// TIA Portal project "Carroponte" (V15.1)

(* hardware
DEVICE "S7-1200 station_1"  S7-1200 Station
   slot 0: "Telaio di montaggio_0"  S7-1200 Rack  Rack  V1.0
   slot 1: "PLC_1"  CPU 1214C DC/DC/DC  6ES7 214-1AG40-0XB0  V4.2
*)

// ===== PLC "PLC_1"  CPU 1214C DC/DC/DC =====

VAR_GLOBAL   // PLC tag table "Tabella delle variabili standard"
   "right" AT %Q0.0 : Bool;
   "left" AT %Q0.1 : Bool;
   "up" AT %Q0.2 : Bool;
   "down" AT %Q0.3 : Bool;
   "start" AT %I0.0 : Bool;
   "s1" AT %I0.1 : Bool;
   "s2" AT %I0.2 : Bool;
   "s3" AT %I0.3 : Bool;
   "sup" AT %I0.4 : Bool;
   "sdown" AT %I0.5 : Bool;
END_VAR

VAR_GLOBAL CONSTANT   // PLC tag table "Tabella delle variabili standard"
   "tempo" : Time := T#5s;
END_VAR

DATA_BLOCK "Variabili_Stato"   // DB1
{ S7_Optimized_Access := 'TRUE' }
VERSION : 0.1
   VAR RETAIN
      home : Bool := true;
   END_VAR
   VAR
      destra1 : Bool;
      su : Bool;
      destra2 : Bool;
      attesa : Bool;
      sinistra : Bool;
      giu : Bool;
   END_VAR
BEGIN
END_DATA_BLOCK

// folder: System blocks/Program resources

DATA_BLOCK "IEC_Timer_0_DB"   // DB2
{ S7_Optimized_Access := 'TRUE' }
AUTHOR : Simatic
FAMILY : IEC
NAME : IEC_TMR
VERSION : 1.0
// stored: InstanceOfName IEC_TIMER
"IEC_TIMER"
BEGIN
END_DATA_BLOCK

// folder: (top level)

ORGANIZATION_BLOCK "Main"   // OB1, LAD, ProgramCycle
TITLE = "Main Program Sweep (Cycle)"
{ S7_Optimized_Access := 'TRUE' }
VERSION : 0.1
   VAR_INPUT
      Initial_Call : Bool;   // Initial call of this OB
      Remanence : Bool;   // =True, if remanent data are available
   END_VAR
BEGIN

REGION Network 1
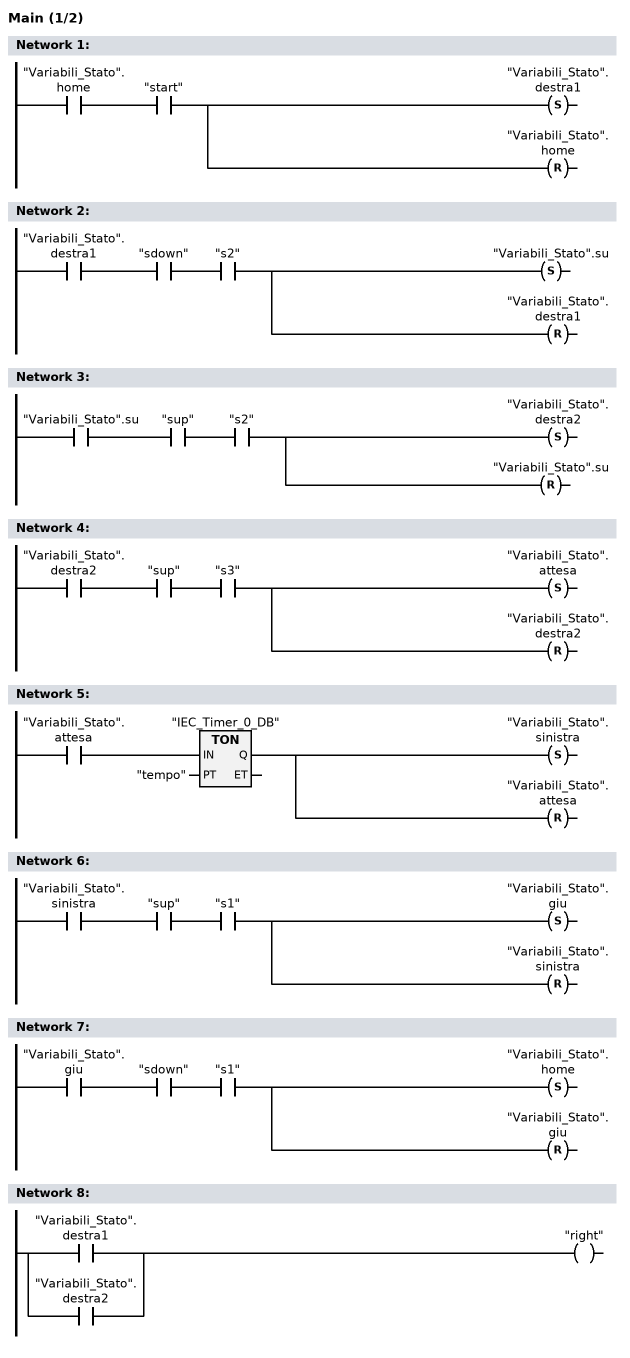
   RUNG wire#powerrail
      Contact( "Variabili_Stato".home )
      Contact( "start" )
      wire#w1
      S_Coil( "Variabili_Stato".destra1 )
   END_RUNG
   RUNG wire#w1
      R_Coil( "Variabili_Stato".home )
   END_RUNG
   // the same network as SCL:
   IF "Variabili_Stato".home AND "start" THEN
       "Variabili_Stato".destra1 := TRUE;
       "Variabili_Stato".home := FALSE;
   END_IF;
END_REGION

REGION Network 2
   RUNG wire#powerrail
      Contact( "Variabili_Stato".destra1 )
      Contact( "sdown" )
      Contact( "s2" )
      wire#w1
      S_Coil( "Variabili_Stato".su )
   END_RUNG
   RUNG wire#w1
      R_Coil( "Variabili_Stato".destra1 )
   END_RUNG
   // the same network as SCL:
   IF "Variabili_Stato".destra1 AND "sdown" AND "s2" THEN
       "Variabili_Stato".su := TRUE;
       "Variabili_Stato".destra1 := FALSE;
   END_IF;
END_REGION

REGION Network 3
   RUNG wire#powerrail
      Contact( "Variabili_Stato".su )
      Contact( "sup" )
      Contact( "s2" )
      wire#w1
      S_Coil( "Variabili_Stato".destra2 )
   END_RUNG
   RUNG wire#w1
      R_Coil( "Variabili_Stato".su )
   END_RUNG
   // the same network as SCL:
   IF "Variabili_Stato".su AND "sup" AND "s2" THEN
       "Variabili_Stato".destra2 := TRUE;
       "Variabili_Stato".su := FALSE;
   END_IF;
END_REGION

REGION Network 4
   RUNG wire#powerrail
      Contact( "Variabili_Stato".destra2 )
      Contact( "sup" )
      Contact( "s3" )
      wire#w1
      S_Coil( "Variabili_Stato".attesa )
   END_RUNG
   RUNG wire#w1
      R_Coil( "Variabili_Stato".destra2 )
   END_RUNG
   // the same network as SCL:
   IF "Variabili_Stato".destra2 AND "sup" AND "s3" THEN
       "Variabili_Stato".attesa := TRUE;
       "Variabili_Stato".destra2 := FALSE;
   END_IF;
END_REGION

REGION Network 5
   "IEC_Timer_0_DB".TON(IN := "Variabili_Stato".attesa, PT := "tempo");
   IF "IEC_Timer_0_DB".Q THEN
       "Variabili_Stato".sinistra := TRUE;
       "Variabili_Stato".attesa := FALSE;
   END_IF;
END_REGION

REGION Network 6
   RUNG wire#powerrail
      Contact( "Variabili_Stato".sinistra )
      Contact( "sup" )
      Contact( "s1" )
      wire#w1
      S_Coil( "Variabili_Stato".giu )
   END_RUNG
   RUNG wire#w1
      R_Coil( "Variabili_Stato".sinistra )
   END_RUNG
   // the same network as SCL:
   IF "Variabili_Stato".sinistra AND "sup" AND "s1" THEN
       "Variabili_Stato".giu := TRUE;
       "Variabili_Stato".sinistra := FALSE;
   END_IF;
END_REGION

REGION Network 7
   RUNG wire#powerrail
      Contact( "Variabili_Stato".giu )
      Contact( "sdown" )
      Contact( "s1" )
      wire#w1
      S_Coil( "Variabili_Stato".home )
   END_RUNG
   RUNG wire#w1
      R_Coil( "Variabili_Stato".giu )
   END_RUNG
   // the same network as SCL:
   IF "Variabili_Stato".giu AND "sdown" AND "s1" THEN
       "Variabili_Stato".home := TRUE;
       "Variabili_Stato".giu := FALSE;
   END_IF;
END_REGION

REGION Network 8
   RUNG wire#powerrail
      Contact( "Variabili_Stato".destra1 )
      wire#w1
      Coil( "right" )
   END_RUNG
   RUNG wire#powerrail
      Contact( "Variabili_Stato".destra2 )
   END_RUNG wire#w1
   // the same network as SCL:
   "right" := "Variabili_Stato".destra1 OR "Variabili_Stato".destra2;
END_REGION

REGION Network 9
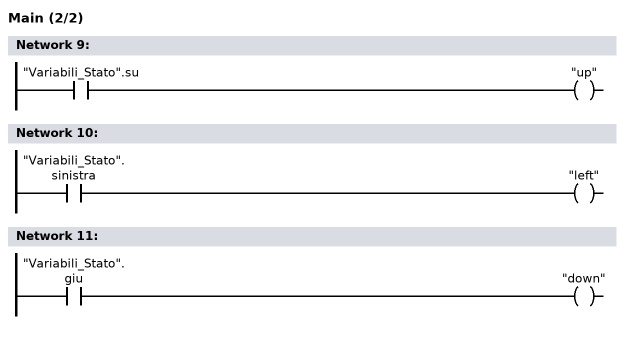
   RUNG wire#powerrail
      Contact( "Variabili_Stato".su )
      Coil( "up" )
   END_RUNG
   // the same network as SCL:
   "up" := "Variabili_Stato".su;
END_REGION

REGION Network 10
   RUNG wire#powerrail
      Contact( "Variabili_Stato".sinistra )
      Coil( "left" )
   END_RUNG
   // the same network as SCL:
   "left" := "Variabili_Stato".sinistra;
END_REGION

REGION Network 11
   RUNG wire#powerrail
      Contact( "Variabili_Stato".giu )
      Coil( "down" )
   END_RUNG
   // the same network as SCL:
   "down" := "Variabili_Stato".giu;
END_REGION
END_ORGANIZATION_BLOCK